{attribute 'call_after_init'}
FUNCTION_BLOCK FINAL UdintParam EXTENDS BaseParam
VAR_INPUT
END_VAR
VAR_OUTPUT
	value: UDINT;
END_VAR
VAR
	
END_VAR

METHOD Change_Param
VAR_INPUT
	value	: STRING;
END_VAR
THIS^.value := STRING_TO_UDINT(value);
_display := UDINT_TO_STRING(THIS^.value);
END_METHOD

METHOD Quick_Change
VAR_INPUT
	value: UDINT;
END_VAR
THIS^.value := value;
_display := UDINT_TO_STRING(THIS^.value);
END_METHOD

END_FUNCTION_BLOCK

(* stored: Version 1.1.0.1, ProductVersion 3.1.4024.12
   POU UdintParam: Id {80291050-3272-447c-b16b-f08de1cfb793}, SpecialFunc None
   Method Change_Param: Id {89a37ef8-e48d-4dde-833c-819f59ec7a37}
   Method Quick_Change: Id {e66f1341-5b5c-4f83-b81c-234669d2057c} *)
